// TIA Portal V16 export
// export: Created 2023-03-29T11:04:39.3049119Z, ExportSetting WithDefaults, DisplayName Totally Integrated Automation Portal, DisplayVersion V16 Update 6, DisplayName TIA Portal Version Control Interface, DisplayVersion V16 Update 2, DisplayName TIA Portal Openness, DisplayVersion V16 Update 6, DisplayName STEP 7 Professional, DisplayVersion V16 Update 6, DisplayName STEP 7 Safety, DisplayVersion V16, DisplayName WinCC Advanced, DisplayVersion V16 Update 6
FUNCTION "Saving_Changed_Data_Word_USint" : Void   // FC65, LAD
{ S7_Optimized_Access := 'TRUE' }
AUTHOR : rtecmer
VERSION : 0.1
// Porównanie czy doszło do zmiany watości w db Hold_RRG <> db HoldRegSlave_toMT101
// stored: AutoNumber false, IsIECCheckEnabled false, SetENOAutomatically false, UDAEnableTagReadback false
   VAR_IN_OUT
      dbHpld_RRG_set : USInt;   // Wartość zadawana porównywana
      dbHoldRegSlave_MT101_inst : Int;   // Wartość do której porównujemy
      memTrig_Client_Receiving : Bool;   // pamiec zbocza zmiany
   END_VAR
   VAR_TEMP   // added for the SCL form of the ladder/FBD networks
      _w1 : Bool;
      _w2 : Bool;
   END_VAR
BEGIN

REGION Network 1
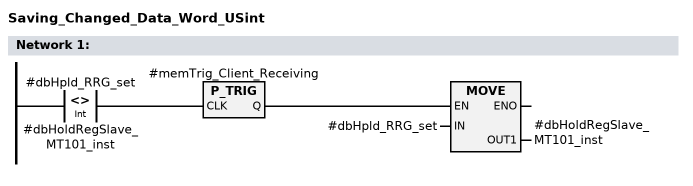
   RUNG wire#powerrail
      { S7_Templates := "SrcType := Int" } NE_Contact(in1 := #dbHpld_RRG_set, in2 := #dbHoldRegSlave_MT101_inst)
      P_Trig( #memTrig_Client_Receiving )
      Move(in := #dbHpld_RRG_set, out1 => #dbHoldRegSlave_MT101_inst)
   END_RUNG
   // the same network as SCL:
   #_w1 := #dbHpld_RRG_set <> #dbHoldRegSlave_MT101_inst;
   #_w2 := #_w1 AND NOT #memTrig_Client_Receiving;   // rising edge
   #memTrig_Client_Receiving := #_w1;
   IF #_w2 THEN #dbHoldRegSlave_MT101_inst := #dbHpld_RRG_set; END_IF;
END_REGION
END_FUNCTION
